# EPICS substitutions: depo-orig/depoApp/Db/TE_TC.substitutions
file TE_TC.template { pattern
{ Sys	, Dev		,PORT		, Chan	}
{ Depo	, "{TTC:1}"	, Depo_TTC1	, 1	}
}
